// Mitsubishi GX Works2 project: Estrutura Condicional   PLC: Q03UDV

// task Task_01 (event TRUE, interval 0, priority 31): POU_01
// task Poll_ST (event TRUE, interval 0, priority 31): Poll_ST

PROGRAM POU_01
VAR
  habilitar : BOOL;
  fTipoOper : STRING[32];
  valor1 : INT;
  valor2 : INT;
  result : INT;
END_VAR
(* structured ladder/FBD written out as ST: instructions are called as NAME(EN, inputs, outputs); _pN, _eN, _tN stand for wires *)
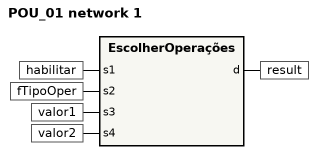
(* network 1 *)
result := EscolherOperações(habilitar, fTipoOper, valor1, valor2);
END_PROGRAM

FUNCTION EscolherOperações
VAR_INPUT
  xHabilitar : BOOL;
  fTipoOper : STRING[32];
  iValor1 : INT;
  iValor2 : INT;
END_VAR
IF xHabilitar THEN
	
	IF fTipoOper="+" THEN
		EscolherOperações:= iValor1+iValor2;
	ELSIF fTipoOper="-" THEN
		EscolherOperações:= iValor1-iValor2;
	ELSIF fTipoOper="*" THEN
		EscolherOperações:= iValor1*iValor2;
	ELSIF fTipoOper="/" THEN
		EscolherOperações:= iValor1/iValor2;
	ELSIF(fTipoOper="M") OR (fTipoOper="m") THEN
		EscolherOperações:= iValor1 MOD iValor2;
	ELSE
		EscolherOperações:= 32767;
	END_IF;
	
	ELSE
	   EscolherOperações:= -32767;
END_IF;
END_FUNCTION

PROGRAM Poll_ST
VAR
  resultado : ARRAY [0..9] OF INT;
END_VAR
resultado[0] :=  EscolherOperações( TRUE , "*" , 2 , 10 );
END_PROGRAM
